FUNCTION_BLOCK itfFaultImplement IMPLEMENTS itfFault
VAR_INPUT
END_VAR
VAR_OUTPUT
END_VAR
VAR
	Fault : BOOL;
	FaultStatus : BOOL;
	ResetButton : BOOL;
END_VAR

METHOD mResetFault : BOOL
IF pResetButton AND NOT pFault THEN
	pFaultStatus := FALSE;
END_IF
END_METHOD

METHOD mSetFault : BOOL
IF pFault THEN
	pFaultStatus := TRUE;
	mSetFault := TRUE;
END_IF
END_METHOD

{warning 'add property implementation'}
PROPERTY pFault : BOOL
GET
pFault := Fault;
END_GET
SET
Fault := pFault;
END_SET
END_PROPERTY

{warning 'add property implementation'}
PROPERTY pFaultStatus : BOOL
GET
pFaultStatus := FaultStatus;
END_GET
SET
FaultStatus := pFaultStatus;
END_SET
END_PROPERTY

{warning 'add property implementation'}
PROPERTY pResetButton : BOOL
GET
pResetButton := ResetButton;
END_GET
SET
ResetButton := pResetButton;
END_SET
END_PROPERTY

END_FUNCTION_BLOCK

(* stored: Version 1.1.0.1, ProductVersion 3.1.4024.12
   POU itfFaultImplement: Id {dfdfd176-5bd6-4f72-8fd3-00022ebdd54e}, SpecialFunc None
   Method mResetFault: Id {757934de-235a-4d3e-9eb8-5f1ed5701c96}
   Method mSetFault: Id {6d3e00e7-868d-4867-928d-29bb036ebb3b}
   Property pFault: Id {3655657d-3612-4f67-ba48-f9919ea50c98}
   Get Get: Id {8f227655-6bd7-4a33-b4b9-6d0b12a41b7c}
   Set Set: Id {500ce595-0f78-4e1d-9349-766ea73d8556}
   Property pFaultStatus: Id {afd11c66-758b-4df2-90a9-4dc789d23088}
   Get Get: Id {0f8f9fa4-e21a-47c8-8155-e980d77e9868}
   Set Set: Id {bcb3c724-9b55-4b0d-be38-b04eb83dfbb2}
   Property pResetButton: Id {19908a86-5193-46bc-af8c-62a2c2eac597}
   Get Get: Id {e51af41c-1455-4bf3-8215-78f1a51a8131}
   Set Set: Id {61366bac-4426-4eb7-bf92-b4a46a75cdc0} *)
